INTERFACE I_Peeker EXTENDS I_Base

METHOD PeekCollection
VAR_INPUT
	Collection : I_Collection;
END_VAR
END_METHOD

END_INTERFACE

(* stored: Version 1.1.0.1, ProductVersion 3.1.4026.18
   Itf I_Peeker: Id {b7429f6b-3d35-4e23-97c7-df9fd385493d}
   Method PeekCollection: Id {c3d81d9a-bba0-40fd-b52a-dec6b604d15e} *)
